Staubli VAL3: Expansion.pjx

--- Expansion.pjx ---
Parameters version=s7.9.1 stackSize=5000 millimeterUnit=true
Program file=copyFile.pgx
Program file=deleteFile.pgx
Program file=fileExit.pgx
Program file=fileRead.pgx
Program file=fileWrite.pgx
Program file=fitCircle.pgx
Program file=getMemoryFree.pgx
Program file=getPwrCnt.pgx
Program file=getState.pgx
Program file=renameFile.pgx
Program file=setLimit.pgx
Program file=start.pgx
Program file=stop.pgx
Data file=Expansion.dtx

--- Expansion.dtx ---
mdesc mNomSpeed
num nState
string sFileDelete = "Disk://data/deletedfile"
string sFrom = "Disk://data/copy/1.txt"
string sTo = "Disk://data/copy/copy.txt"
string sFromRename = "Disk://data/rename/1.txt"
string sToRename = "Disk://data/rename/re.txt"
string sFileExist = "Disk://data/exist/exist.txt"
string sFileRead = "Disk://data/fileoperation/read.txt"
num nFileHandler
num nLine
string sLine
string sFileWrite = "Disk://data/fileoperation/write.txt"
num nPwrCnt
num nCircleErr
pointRx pPointIn[4]
  [0] = {fatherId=world[0]}
  [1] = {fatherId=world[0]}
  [2] = {fatherId=world[0]}
  [3] = {fatherId=world[0]}
num nRadius
frame fCircleFrame = {fatherId=world[0]}
jointRx jArmLimit[2]
  [0] = {j1=-100, j2=-50, j3=-50, j4=-100, j5=-60, j6=-100}
  [1] = {j1=150, j2=100, j3=100, j4=100, j5=100, j6=100}
jointRx jCellLimit[2]
  [0] = {j1=-100, j2=-100, j3=-100, j4=-100, j5=-85, j6=-100}
  [1] = {j1=120, j2=120, j3=120, j4=120, j5=90, j6=300}

--- start.pgx ---
program start()
begin
  //Here are examples for expansion addon functions.

  //
  title("Expansion examples")
  userPage()
  cls()
  //$getState
  call getState()
  //$delete
  call deleteFile()
  //$copy
  call copyFile()
  //$rename
  call renameFile()
  //$fileExists
  call fileExit()
  //$fileGet
  call fileRead()
  //$fileSet
  call fileWrite()
  //$getPowerCount
  call getPwrCnt()
  //$getFreeSpace
  call getMemoryFree()
  //$circleFind
  call fitCircle()
  //$setArmLimit,$setCellLimit
  call setLimit()
end

--- copyFile.pgx ---
program copyFile()
  local bool l_bRes
begin
  //copy file or folder from sFrom to sTo
  l_bRes=$copy(sFrom,sTo)
  if l_bRes
    gotoxy(1,3)
    put("拷贝文件:"+sFrom+"至"+sTo)
  else
    gotoxy(1,3)
    put("拷贝文件出错:"+sFrom)
  endIf

end

--- deleteFile.pgx ---
program deleteFile()
  local bool l_bRes
begin
  //delete the file or folder
  l_bRes=$delete(sFileDelete)
  if l_bRes
    gotoxy(1,2)
    put("删除:"+sFileDelete)
  else
    gotoxy(1,2)
    put("删除:失败"+sFileDelete)
  endIf

end

--- fileExit.pgx ---
program fileExit()
  local bool l_bRes
begin
  //
  l_bRes=$fileExists(sFileExist)
  if l_bRes
    gotoxy(1,7)
    put("文件存在:"+sFileExist)
  else
    gotoxy(1,7)
    put("文件不存在:"+sFileExist)
  endIf

end

--- fileRead.pgx ---
program fileRead()
  local bool l_bRes
begin
  //file operation:open ,read, write,close
  //
  l_bRes=$fileExists(sFileRead)
  if !l_bRes
    popUpMsg("文件不存在："+sFileRead)
    return
  endIf
  //防止某个文件没有关闭
  $fileClose(0)
  $fileClose(1)
  $fileClose(2)
  $fileClose(3)
  $fileClose(4)
  $fileClose(5)
  $fileClose(6)
  $fileClose(7)
  $fileClose(8)
  $fileClose(9)
  //以读取（r）的方式打开文件
  nFileHandler=$fileOpen(sFileRead,"r")
  if nFileHandler<0 or nFileHandler>9
    popUpMsg("打开文件失败："+sFileRead)
    return
  endIf

  do
      //每次读取一行,当然可以读取多行，sLine大小和读取行数最好一致。
      nLine=$fileGet(nFileHandler,sLine,1)
      //这里可以放置处理读取内容的代码
      //
      //
      delay(0)
    until nLine<=0


    //达到文件末尾或其他跳出文件读取时，必须关闭文件
    $fileClose(nFileHandler)
    //
end

--- fileWrite.pgx ---
program fileWrite()
  local bool l_bRes
  local num l_nCount
begin
  //file operation:open ,read, write,close
  //
  l_bRes=$fileExists(sFileWrite)
  if !l_bRes
    popUpMsg("文件不存在："+sFileWrite)
    return
  endIf
  //防止某个文件没有关闭
  $fileClose(0)
  $fileClose(1)
  $fileClose(2)
  $fileClose(3)
  $fileClose(4)
  $fileClose(5)
  $fileClose(6)
  $fileClose(7)
  $fileClose(8)
  $fileClose(9)
  //以读取（w）的方式打开文件
  nFileHandler=$fileOpen(sFileWrite,"w")
  if nFileHandler<0 or nFileHandler>9
    popUpMsg("打开文件失败："+sFileWrite)
    return
  endIf
  //写入文件，这里以计数方式结束写入，当然可以使用用户自定义结束。
  //写入文件结束是必须的，否则会造成系统瘫痪。
  l_nCount=0
  sLine="a"
  do
    //每次写入一行,当然可以写入多行，sLine大小和写入行数最好一致。
    nLine=$fileSet(nFileHandler,sLine,1)
    l_nCount=l_nCount+1
    //
    delay(0)
  until l_nCount>500


  //达到文件末尾或其他跳出文件读取时，必须关闭文件
  $fileClose(nFileHandler)
  //
end

--- fitCircle.pgx ---
program fitCircle()
begin
  //fit a circle through pPointIn array.
  nCircleErr=$circleFind(pPointIn,fCircleFrame,nRadius)
  if nCircleErr<0
    gotoxy(1,10)
    put("圆:拟合失败！")
    return
  endIf
  gotoxy(1,10)
  put("圆半径："+toString(".2",nRadius)+"  "+"误差："+toString(".2",nCircleErr))
end

--- getMemoryFree.pgx ---
program getMemoryFree()
  local num l_nSpace
begin
  //
  l_nSpace=$getFreeSpace("/usr")
  gotoxy(1,9)
  put("sys free space:"+toString(".2",l_nSpace))
end

--- getPwrCnt.pgx ---
program getPwrCnt()
begin
  //
  nPwrCnt=$getPowerCount()
  gotoxy(1,8)
  put("总上电小时数："+toString("",nPwrCnt))
end

--- getState.pgx ---
program getState()
begin
  nState=$getState()
  gotoxy(1,1)
  put("RSI state:"+toString("",nState)+"   ")
end

--- renameFile.pgx ---
program renameFile()
  local bool l_bRes
begin
  //rename file or folder
  l_bRes=$rename(sFromRename,sToRename)
  if l_bRes
    gotoxy(1,5)
    put("更名："+sFromRename+"至"+sToRename)
  else
    gotoxy(1,5)
    put("更名失败："+sFromRename+"至"+sToRename)
  endIf
end

--- setLimit.pgx ---
program setLimit()
  local bool l_bRes
begin
  //set arm/cell limit:
  //
  l_bRes=$setArmLimits(jArmLimit[0],jArmLimit[1])
  if l_bRes
    gotoxy(1,11)
    put("setArmLimit:OK")
  else
    gotoxy(1,11)
    put("setArmLimit:fail")
  endIf
  //
  l_bRes=$setArmLimits(jCellLimit[0],jCellLimit[1])
  if l_bRes
    gotoxy(20,11)
    put("setCellLimit:OK")
  else
    gotoxy(20,11)
    put("setCellLimit:fail")
  endIf
end
